(*
	RJM Maszyny sp. z o.o.
	autor 	: Rafał Osajda
	data	: 02.02.2024
	TC		: 3.1 4024.54
	wersja	: 0.0.1.0	: pełna obsługa

	Obsługa elektrozaworu do sterowania siłownikiem pneumatycznym.sterowanie 5 na 2 1 cewka
*)
FUNCTION_BLOCK FB_Elektrozawor_5na2_1Cewka EXTENDS FB_Electrovalve

METHOD FB_init : BOOL
VAR_INPUT
	bInitRetains : BOOL; // if TRUE, the retain variables are initialized (warm start / cold start)
	bInCopyCode : BOOL;  // if TRUE, the instance afterwards gets moved into the copy code (online change)
END_VAR
THIS^.eRodzaj			:= E_ElectrovalveType.C1_5na2;
END_METHOD

(*
	RJM Maszyny sp. z o.o.
	autor 	: Rafał Osajda
	data	: 21.02.2024
	TC		: 3.1 4024.54
	wersja	: 0.0.1.0	: pełna obsługa

	Ustawienie odpowiednich wyjść
*)
METHOD Steruj : BOOL
VAR_INPUT
	eAkcja	: E_ElectrovalveAction;
END_VAR
CASE eAkcja OF
	E_ElectrovalveAction.e_EL_Wyj4_Wylacz	:
		bCewkaA								:= FALSE;
	E_ElectrovalveAction.e_EL_Wyj4_Wlacz	:
		bCewkaA								:= TRUE;
	E_ElectrovalveAction.e_EL_DoPoczatku	:
		bCewkaA								:= FALSE;
	E_ElectrovalveAction.e_EL_DoKonca		:
		bCewkaA								:= TRUE;
	E_ElectrovalveAction.e_EL_Reset			:
		bCewkaA								:= FALSE;
END_CASE
THIS^.bCewkaB								:= FALSE;
END_METHOD

END_FUNCTION_BLOCK

(* stored: Version 1.1.0.1
   POU FB_Elektrozawor_5na2_1Cewka: Id {f05beb48-ad03-02a9-17e7-b14c81a9cbb4}, SpecialFunc None
   Method FB_init: Id {6b3bf50e-cc11-4a3c-99c4-2a04d7452798}
   Method Steruj: Id {51b0d103-b3ed-080b-10c4-25225c130a03} *)
